(* CoDeSys 2.3.9.36 project: KVR_Mast.1.3.pro *)
(* Version: 13 *)
(* Author: JB *)
(* Libraries: ifm_CR0401\ifm_CR0401_V030100.lib 30.7.20 09:49:34, ifm_RAWCan\ifm_RAWCan_NT_V020004.lib 27.10.21 17:23:48, ifm_CANopen\ifm_CANopen_NT_V020004.lib 27.10.21 17:23:48, ifm_CANopen\3S_CanDrv.lib 27.10.21 17:23:48, ifm_CANopen\3S_CANopenManager.lib 27.10.21 17:23:48, Util.lib 6.11.07 14:39:24, standard.lib 4.10.05 11:14:46, SysLibCallback.lib 26.9.08 16:43:52 *)

(* PLC configuration (modules and I/O channels)
Configuration [LocalConfiguration] node 0, in %IB0 out %QB0 {IFM_PARAM_WORD_TIME = 0}
Input/Output [LocalInputOutput] node 1, in %IB0 out %QB0
IN00 AT %IB0 [ChInputBool] Input 00 Bit
IN01 AT %IB1 [ChInputBool] Input 01 Bit
IN02 AT %IB2 [ChInputBool] Input 02 Bit
IN03 AT %IB3 [ChInputBool] Input 03 Bit
IN04 AT %IB4 [ChInputBool] Input 04 Bit
IN05 AT %IB5 [ChInputBool] Input 05 Bit
IN06 AT %IB6 [ChInputBool] Input 06 Bit
IN07 AT %IB7 [ChInputBool] Input 07 Bit
IN08 AT %IB8 [ChInputBool] Input 08 Bit
IN09 AT %IB9 [ChInputBool] Input 09 Bit
IN10 AT %IB10 [ChInputBool] Input 10 Bit
IN11 AT %IB11 [ChInputBool] Input 11 Bit
OUT00 AT %QB0 [ChOutputBool] Output 00 Bit
OUT01 AT %QB1 [ChOutputBool] Output 01 Bit
OUT02 AT %QB2 [ChOutputBool] Output 02 Bit
OUT03 AT %QB3 [ChOutputBool] Output 03 Bit
OUT04 AT %QB4 [ChOutputBool] Output 04 Bit
OUT05 AT %QB5 [ChOutputBool] Output 05 Bit
OUT06 AT %QB6 [ChOutputBool] Output 06 Bit
OUT07 AT %QB7 [ChOutputBool] Output 07 Bit
System Inputs [LocalSystemInputs] node 2, in %IB12 out %QB8
  SUPPLY_VOLTAGE_VBBS AT %IW6 [ChInputWord] Supply voltage VBBS
  SUPPLY_VOLTAGE_VU AT %IW7 [ChInputWord] Supply voltage VU
  SUPPLY_VOLTAGE_VBB1 AT %IW8 [ChInputWord] Supply voltage VBB1
  SUPPLY_VOLTAGE_VBB2 AT %IW9 [ChInputWord] Supply voltage VBB2
  TEMPERATURE AT %IW10 [ChInputInt] Temperature
J1939 Interface [CAN_J1939] node 1, in %IB22 out %QB8
J1939 Interface [CAN_J1939] node 1, in %IB44 out %QB16
*)

(* Global variable list: Global_Constants *)
VAR_GLOBAL CONSTANT

	MAX_CTRLINDEX: BYTE := 0;

	SIMULATIONSMODUS: BOOL := FALSE;

	(* Flag positions for variable FlagsECU2PC *)
	ECU2PC_AllowRemote: INT := 3;
	ECU2PC_EmergencyStop: INT := 4;
	ECU2PC_RemoteAckn: INT := 6;
	ECU2PC_MainSwitch: INT := 7;

	(* Flag positions for variable FlagsPC2ECU *)
	PC2ECU_Remote: INT := 0;
	PC2ECU_BlackOut: INT := 1;
	PC2ECU_ResetMotorActiveTime: INT := 3;

	(* Flag positions for variables Mast[x].FlagsECU2PC *)
	ECU2PC_TopPosition: INT := 0;
	ECU2PC_BottomPosition: INT := 1;
	ECU2PC_MovingUp: INT := 2;
	ECU2PC_MovingDown: INT := 3;
	ECU2PC_LocalUp: INT := 4;
	ECU2PC_LocalDown: INT := 5;
	ECU2PC_LimitSwitch4m: INT := 7;
	ECU2PC_LimitSwitchBottom: INT := 8;
	ECU2PC_NotReadyToSwitchOn: INT := 9;
	ECU2PC_ParkPosition: INT := 10;
	ECU2PC_MontagePos: INT := 11;
	ECU2PC_LimitSwitchAufgerichtet: INT := 12;

	(* Flag positions for variables Mast[x].FlagsPC2ECU *)
	PC2ECU_MoveUp: INT := 0;
	PC2ECU_MoveDown: INT := 1;
	PC2ECU_SlowSpeed: INT := 2;

	(* Flag positions for variable Mast[x].ErrorECU2PC *)
	ECU2PC_ErrorFU: INT 					:= 0;
	ECU2PC_ErrorCanTimeout: INT 			:= 1;
	ECU2PC_ErrorMastSchrittkette: INT 		:= 4;

	QSCMD_NOP: BYTE				:= 0;
	QSCMD_CLEAR_ERROR: BYTE		:= 1;
	QSCMD_QUICK_STOP: BYTE		:= 113;
	QSCMD_HALT: BYTE			:= 114;
	QSCMD_VELOCITY_MODE: BYTE	:= 117; (* QSData0 = desired velocity *)
	QSCMD_ABS_POS_MODE: BYTE	:= 118; (* QSData0 = desired velocity, QSData1 = desired position *)

	(* Flag positions for FU statusword *)
	STAT_ENABLED: INT			:= 0;
	STAT_ERROR: INT				:= 1;
	STAT_WARNING: INT			:= 2;
	STAT_MOVING: INT			:= 3;
	STAT_REACHED: INT			:= 4;
	STAT_LIMIT: INT				:= 5;
	STAT_STOP_OR_HALT: INT		:= 11;

	FU1_POS_TO_MM: REAL 		:= 4.1114E-004;

	CAN_CHANNEL_HOST: BYTE 		:= 1;
	CAN_CHANNEL_LOCAL: BYTE 	:= 2;

	FU1_NODE_ID: BYTE			:= 127;

	MAX_CURRENT_HIST: WORD		:= 100;
	MAX_ERRORCODE_HIST: BYTE	:= 10;

END_VAR

(* Global variable list: Global_Variables *)
VAR_GLOBAL

	BlinkSlow: BOOL;

	MasterPresent: BOOL;

	inputs: TYPE_INPUTS;
	outputs: TYPE_OUTPUTS;

	canNodeFU1Present: BOOL;

	tasteAuf: BOOL;
	tasteAb: BOOL;
	tasteReset: BOOL;

	FlagsECU2PC: WORD			{parameter list=proc_vars_ecu [name=FlagsECU2PC 					index=16#3000 subindex=1 accessright="read only"] };
	FlagsPC2ECU: WORD			{parameter list=proc_vars_ecu [name=FlagsPC2ECU 					index=16#3000 subindex=2 accessright="write only"] };
	Windspeed: BYTE				{parameter list=proc_vars_ecu [name=Windspeed	 					index=16#3000 subindex=3 accessright="read only"] };
	CabinetTemperature: SINT	{parameter list=proc_vars_ecu [name=Temperature	 					index=16#3000 subindex=4 accessright="read only"] };
	ExtTemperature: SINT		{parameter list=proc_vars_ecu [name=ExtTemperature	 				index=16#3000 subindex=5 accessright="read only"] };
	IntVoltage: WORD			{parameter list=proc_vars_ecu [name=IntVoltage		 				index=16#3000 subindex=6 accessright="read only"] };

	Mast1Height: WORD			{parameter list=proc_vars_mast1 [name=Mast1Height 					index=16#3001 subindex=1 accessright="read only"] };
	Mast1FlagsECU2PC: WORD		{parameter list=proc_vars_mast1 [name=Mast1FlagsECU2PC 				index=16#3003 subindex=1 accessright="read only"] };
	Mast1FlagsPC2ECU: WORD		{parameter list=proc_vars_mast1 [name=Mast1FlagsPC2ECU 				index=16#3004 subindex=1 accessright="write only"] };
	Mast1Current: DINT			{parameter list=proc_vars_mast1 [name=Mast1Current 					index=16#3006 subindex=1 accessright="read only"] };
	Mast1ErrorECU2PC: WORD		{parameter list=proc_vars_mast1 [name=Mast1ErrorECU2PC				index=16#300D subindex=1 accessright="read only"] };
	Mast1FUErrorCode: WORD		{parameter list=proc_vars_mast1 [name=Mast1FUErrorCode				index=16#3010 subindex=1 accessright="read only"] };
	Mast1State: BYTE			{parameter list=proc_vars_mast1 [name=Mast1State					index=16#3012 subindex=1 accessright="read only"] };
	Mast1Speed: DINT			{parameter list=proc_vars_mast1 [name=Mast1Speed					index=16#3013 subindex=1 accessright="read only"] };

	(*
	Mast1TempPcbPower: WORD		{parameter list=proc_vars_mast1 [name=Mast1TempPcbPower				index=16#300A subindex=1 accessright="read only"] };
	Mast1TempPcbController: WORD{parameter list=proc_vars_mast1 [name=Mast1TempPcbController		index=16#300B subindex=1 accessright="read only"] };
	Mast1TempPcbAmplifier: WORD	{parameter list=proc_vars_mast1 [name=Mast1TempPcbAmplifier			index=16#300F subindex=1 accessright="read only"] };
	*)

	Mast1SetEncoderPW: DWORD	{parameter list=Parameters 		[name=Mast1SetEncoderPW				index=16#2014 subindex=1 accessright="read-write"] };

	Version: BYTE				{parameter list=version_info 	[name=Version						index=16#3020 subindex=1 accessright="read only"] };
	VersionDate: DWORD			{parameter list=version_info 	[name=VersionDate					index=16#3020 subindex=2 accessright="read only"] };

	Mast1MotorActiveTimeSeconds2: DWORD {parameter list=proc_vars_mast1 [name=Mast1MotorActiveTimeSeconds2 index=16#3014 subindex=1 accessright="read only"] };

	FU1_Current_Sim: DINT;

	FU1_Current_Hist: ARRAY[0..MAX_CURRENT_HIST] OF DINT;
	FU1_ErrorCode_Idx: BYTE;
	FU1_ErrorCode_Hist: ARRAY[0..MAX_ERRORCODE_HIST] OF INT;

END_VAR

VAR_GLOBAL RETAIN
	Mast1HeightRetain: WORD;
    NullfahrtErforderlich: BOOL;
END_VAR

(* Global variable list: Parameters *)
VAR_GLOBAL RETAIN
	SettingsPW: DWORD := 0	 					{parameter list=Parameters [name=SettingsPW					 	index=16#2000 subindex=12 accessright="read-write"] };
	(* 9000 *)
	Mast1TopPosition: WORD := 12000 				{parameter list=Parameters [name=Mast1TopPosition 				index=16#2006 subindex=1 accessright="read-write"] };
	Mast1BottomPosition: WORD := 2975			{parameter list=Parameters [name=Mast1BottomPosition			index=16#2007 subindex=1 accessright="read-write"] };
	Mast1VelocityNormal: INT := 2500			{parameter list=Parameters [name=Mast1VelocityNormal			index=16#200A subindex=1 accessright="read-write"] };
	Mast1VelocitySlow: INT := 500				{parameter list=Parameters [name=Mast1VelocitySlow				index=16#200B subindex=1 accessright="read-write"] };
	Mast1VelocityBottom: INT := 500				{parameter list=Parameters [name=Mast1VelocityBottom			index=16#200C subindex=1 accessright="read-write"] };
	Mast1BottomPositionOffset: WORD := 60		{parameter list=Parameters [name=Mast1BottomPositionOffset		index=16#200D subindex=1 accessright="read-write"] };
	Mast1CurrentLimitBottom: INT := 30			{parameter list=Parameters [name=Mast1CurrentLimitBottom		index=16#200E subindex=1 accessright="read-write"] };
	Mast1BottomLimitSwitchWindow: WORD := 50	{parameter list=Parameters [name=Mast1BottomLimitSwitchWindow	index=16#200F subindex=1 accessright="read-write"] };
	Mast1MontagePos: WORD := 3975 				{parameter list=Parameters [name=Mast1MontagePos 				index=16#2010 subindex=1 accessright="read-write"] };
	Mast1MotorActiveTimeSeconds: DWORD := 0		{parameter list=Parameters [name=Mast1MotorActiveTimeSeconds	index=16#2013 subindex=1 accessright="read-write"] };
	Mast1CurrentLimit: INT := 50				{parameter list=Parameters [name=Mast1CurrentLimit				index=16#2018 subindex=1 accessright="read-write"] };
	Mast1TopSettlingOffset: INT := 40			{parameter list=Parameters [name=Mast1TopSettlingOffset			index=16#2019 subindex=1 accessright="read-write"] };
END_VAR

(* Data type *)
TYPE TYPE_INPUTS :
	STRUCT
		TasteAusfahren: BOOL;
		TasteEinfahren: BOOL;
		TastePoweredByGenerator: BOOL;
		EndschalterNotantrieb: BOOL;
		EndschalterEingefahren: BOOL;
		EndschalterAufgerichtet: BOOL;
	END_STRUCT
END_TYPE

(* Data type *)
TYPE TYPE_OUTPUTS :
	STRUCT
		LEDAusgefahren: BOOL;
		LEDEingefahren: BOOL;
		LEDMontagePos: BOOL;
		RelaisMotorLeistung: BOOL;
		SchuetzGrundlast: BOOL;
	END_STRUCT
END_TYPE

(* POU PLC_PRG, FBD *)
PROGRAM PLC_PRG
VAR
	Init1: BOOL:=TRUE;
	CycleTime:DWORD;
	MaxCycleTime:DWORD;
	ResetMax:BOOL;
END_VAR
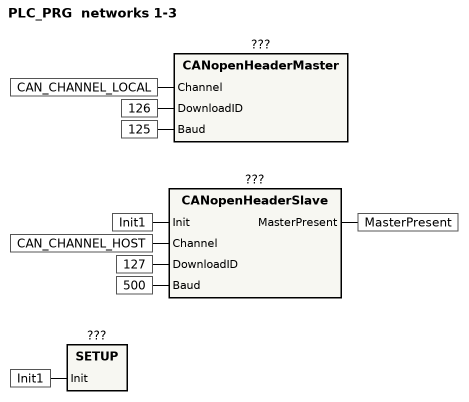
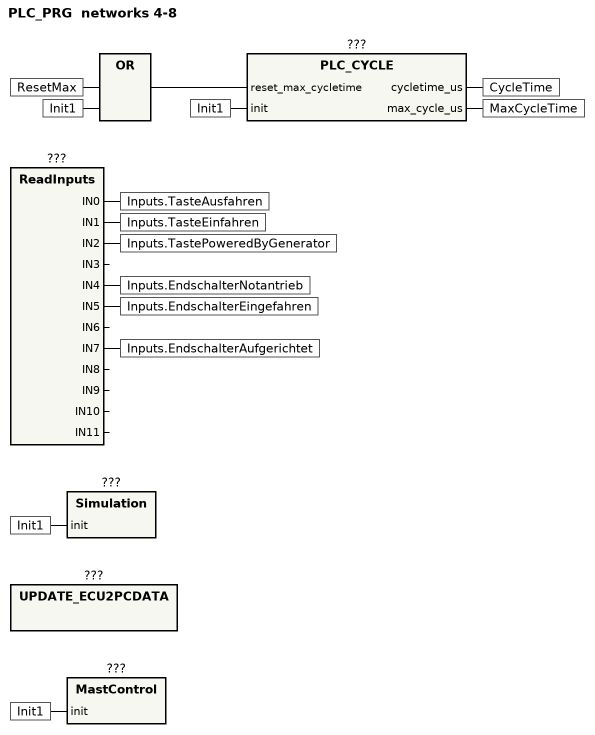
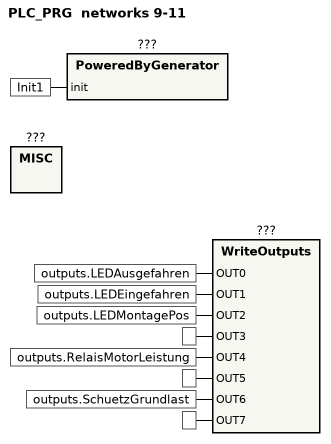
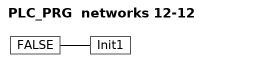
_FBD_ (* Function Block Diagram *)
NETWORK 1 (* CAN Master auf CAN2 initialisieren (Schnittstelle zu FU) *)
	???:CANopenHeaderMaster(Channel: CAN_CHANNEL_LOCAL, DownloadID: 126, Baud: 125)
NETWORK 2 (* CAN Slave auf CAN1 initialisieren (Schnittstelle zu PC) *)
	???:CANopenHeaderSlave(Init: Init1, Channel: CAN_CHANNEL_HOST, DownloadID: 127, Baud: 500) => MasterPresent
NETWORK 3
	???:SETUP(Init: Init1)
NETWORK 4
	???:PLC_CYCLE(reset_max_cycletime: OR(ResetMax, Init1), init: Init1, max_cycle_us => MaxCycleTime) => CycleTime
NETWORK 5
	???:ReadInputs(IN1 => Inputs.TasteEinfahren, IN2 => Inputs.TastePoweredByGenerator, IN4 => Inputs.EndschalterNotantrieb, IN5 => Inputs.EndschalterEingefahren, IN7 => Inputs.EndschalterAufgerichtet) => Inputs.TasteAusfahren
NETWORK 6
	???:Simulation(init: Init1)
NETWORK 7
	???:UPDATE_ECU2PCDATA()
NETWORK 8
	NOT ???:MastControl(init: Init1)
NETWORK 9
	???:PoweredByGenerator(init: Init1)
NETWORK 10
	???:MISC()
NETWORK 11
	???:WriteOutputs(OUT0: outputs.LEDAusgefahren, OUT1: outputs.LEDEingefahren, OUT2: outputs.LEDMontagePos, OUT3: , OUT4: outputs.RelaisMotorLeistung, OUT5: , OUT6: outputs.SchuetzGrundlast, OUT7: )
NETWORK 12 (* last line *)
	FALSE => Init1
_END_FBD_
(* the same logic as Structured Text *)
(* Network 1: see the listing above *)
(* Network 2: see the listing above *)
(* Network 3: see the listing above *)
(* Network 4: see the listing above *)
(* Network 5: see the listing above *)
(* Network 6: see the listing above *)
(* Network 7: see the listing above *)
(* Network 8: see the listing above *)
(* Network 9: see the listing above *)
(* Network 10: see the listing above *)
(* Network 11: see the listing above *)
(* Network 12 *)
Init1 := FALSE;
END_PROGRAM

(* POU CANopen/CANopenHeaderMaster, FBD *)
PROGRAM CANopenHeaderMaster
VAR_INPUT
	Channel: BYTE;
	DownloadID: BYTE;
	Baud: WORD;
END_VAR
VAR
	(*CAN settings*)
	SettingsCAN: CAN_SETTING_ST;

	(*Set CANopen state*)
	SetCanOpenState: CANOPEN_SETSTATE;
	SetState:BOOL:=TRUE;

	(*Handling CANopen status*)
	HandlingCANopen: CANopen_HANDLING_ST;
	Baudrate: DWORD;
	MasterState: BYTE;
	GuardError: BOOL;
	ErrorNodeList: ARRAY[0..MAXGUARDERR] OF BYTE;
	CanState: BYTE;
	Nodestate: BYTE;
	LastNodeState: BYTE;

	(*Emergency handling*)
	CanEmcy: CAN_EMCY;
	RestEmcyList: BOOL;
	EMCY_MSG_Count: DWORD; (* No of EMCY messages  Leaving errors are count too *)
	EmcyStruct: ARRAY[0..10] OF tT_EMCY;

	(*Handling CAN status*)
	StatusCan: CAN_Status_and_Errors;
	ResetCanFlags: BOOL;
	BusLoad: BYTE;
	BusOff: BOOL;
	RxOverflow: BOOL;
	RxWarning: BOOL;
	TxOverflow: BOOL;
	TxWarning: BOOL;

	GetstateSlave1: CANopen_GetStateSlave;

END_VAR
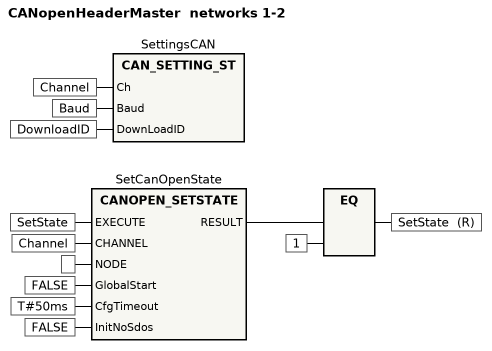
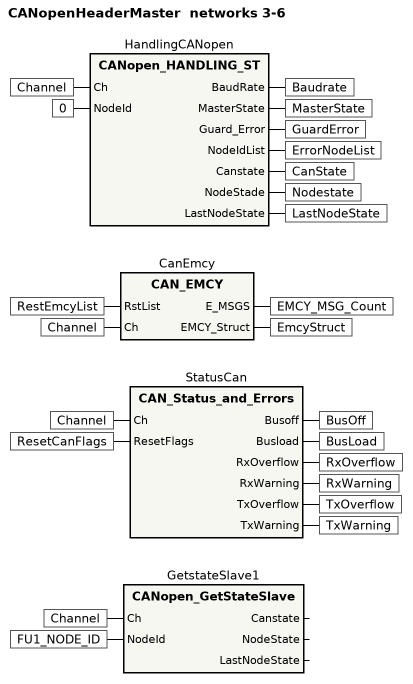
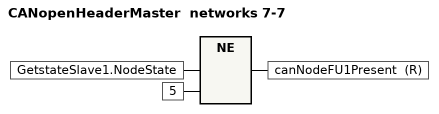
_FBD_ (* Function Block Diagram *)
NETWORK 1 (* Basic functions for the CAN / CANopen functionality *)
	SettingsCAN:CAN_SETTING_ST(Ch: Channel, Baud: Baud, DownLoadID: DownloadID)
NETWORK 2 (* Set CANopen status *)
	EQ(SetCanOpenState:CANOPEN_SETSTATE(EXECUTE: SetState, CHANNEL: Channel, NODE: , GlobalStart: FALSE, CfgTimeout: T#50ms, InitNoSdos: FALSE), 1) => R SetState
NETWORK 3 (* CANopen Master and heartbeat handling *)
	HandlingCANopen:CANopen_HANDLING_ST(Ch: Channel, NodeId: 0, MasterState => MasterState, Guard_Error => GuardError, NodeIdList => ErrorNodeList, Canstate => CanState, NodeStade => Nodestate, LastNodeState => LastNodeState) => Baudrate
NETWORK 4 (* CANopen Emergency Handling for 11 emergency messages *)
	CanEmcy:CAN_EMCY(RstList: RestEmcyList, Ch: Channel, EMCY_Struct => EmcyStruct) => EMCY_MSG_Count
NETWORK 5 (* Get the CAN Status and CAN Errors *)
	StatusCan:CAN_Status_and_Errors(Ch: Channel, ResetFlags: ResetCanFlags, Busload => BusLoad, RxOverflow => RxOverflow, RxWarning => RxWarning, TxOverflow => TxOverflow, TxWarning => TxWarning) => BusOff
NETWORK 6
	GetstateSlave1:CANopen_GetStateSlave(Ch: Channel, NodeId: FU1_NODE_ID)
NETWORK 7
	NE(GetstateSlave1.NodeState, 5) => R canNodeFU1Present
_END_FBD_
(* the same logic as Structured Text *)
(* Network 1 *)
SettingsCAN(Ch := Channel, Baud := Baud, DownLoadID := DownloadID);
(* Network 2: see the listing above *)
(* Network 3 *)
HandlingCANopen(Ch := Channel, NodeId := 0);
MasterState := HandlingCANopen.MasterState;
GuardError := HandlingCANopen.Guard_Error;
ErrorNodeList := HandlingCANopen.NodeIdList;
CanState := HandlingCANopen.Canstate;
Nodestate := HandlingCANopen.NodeStade;
LastNodeState := HandlingCANopen.LastNodeState;
Baudrate := HandlingCANopen.BaudRate;
(* Network 4 *)
CanEmcy(RstList := RestEmcyList, Ch := Channel);
EmcyStruct := CanEmcy.EMCY_Struct;
EMCY_MSG_Count := CanEmcy.E_MSGS;
(* Network 5 *)
StatusCan(Ch := Channel, ResetFlags := ResetCanFlags);
BusLoad := StatusCan.Busload;
RxOverflow := StatusCan.RxOverflow;
RxWarning := StatusCan.RxWarning;
TxOverflow := StatusCan.TxOverflow;
TxWarning := StatusCan.TxWarning;
BusOff := StatusCan.Busoff;
(* Network 6 *)
GetstateSlave1(Ch := Channel, NodeId := FU1_NODE_ID);
(* Network 7 *)
IF GetstateSlave1.NodeState <> 5 THEN canNodeFU1Present := FALSE; END_IF;
END_PROGRAM

(* POU CANopen/CAN_SETTING_ST, ST *)
FUNCTION_BLOCK CAN_SETTING_ST
(* Basic functions for the CAN / CANopen functionality *)
VAR

	CAN_SETDOWNLOADID_: CAN_SETDOWNLOADID;
	CAN_ENABLE_: CAN_ENABLE;
	CANOPEN_ENABLE_: CANOPEN_ENABLE;

	CANOPEN_SETSTATE_: CANOPEN_SETSTATE;
END_VAR
VAR_INPUT
	Ch: BYTE;
	Baud:WORD;
	DownLoadID:BYTE;
END_VAR
CAN_SETDOWNLOADID_(EXECUTE:=TRUE , CHANNEL:=Ch , DOWNLOAD_ID:=DownLoadID , RESULT=> );
CAN_ENABLE_(ENABLE:=TRUE , CHANNEL:=Ch , BAUDRATE:=Baud , RESULT=> );
CANOPEN_ENABLE_(ENABLE:=TRUE , CHANNEL:=Ch , Baudrate:=Baud , RESULT=> );
END_FUNCTION_BLOCK

(* POU CANopen/CANopen_HANDLING_ST, ST *)
FUNCTION_BLOCK CANopen_HANDLING_ST
(* CANopen Master and heartbeat handling *)
VAR
	CANOPEN_GETSTATE_: CANOPEN_GETSTATE;
	Execute_Getstate: BOOL := TRUE;
	CANOPEN_GETGUARDHBERRLIST_: CANOPEN_GETGUARDHBERRLIST;
	Execute_Guardlst: BOOL := TRUE;
	ResetErrorList: BOOL;
	PlcNodeId: BYTE;
	i: INT;
	GuardErrorCnt: WORD;
END_VAR
VAR_INPUT
	Ch: BYTE;
	NodeId: BYTE;
END_VAR
VAR_OUTPUT
	BaudRate: DWORD;
	MasterState: BYTE;
	Guard_Error: BOOL;
	NodeIdList: ARRAY[0..MAXGUARDERR] OF BYTE;
	Canstate: BYTE;
	NodeStade: BYTE;
	LastNodeState: BYTE;
END_VAR
(* ^^^^ Get the current state of the CANopen master ^^^^ *)
CANOPEN_GETSTATE_(
	EXECUTE:=Execute_Getstate ,
	CHANNEL:=Ch ,
	NODE:=NodeId ,
	MASTERSTATE=>MasterState ,
	PLCNODEID=>PlcNodeId ,
	PLCBAUDRATE=>BaudRate ,
	PLCVERSION=>,
	CANSTATE=>Canstate ,
	NODESTATE=>NodeStade ,
	LASTNODESTATE=>LastNodeState ,
	RESULT=> );

(* Values are valid now, function call can be stopped *)
IF CANOPEN_GETSTATE_.RESULT= 1 THEN
	Execute_Getstate:=FALSE;
END_IF

(* Function is passive, execute again *)
IF CANOPEN_GETSTATE_.RESULT= 0 THEN
	Execute_Getstate:=TRUE;
END_IF

(* ^^^^^ Get heartbeaterror or nodeguarding error ^^^^ *)
CANOPEN_GETGUARDHBERRLIST_(
	EXECUTE:=Execute_Guardlst ,
	CHANNEL:=Ch ,
	ResetList:=ResetErrorList ,
	N_NODES=>GuardErrorCnt,
	NODEID=>NodeIdList ,
	RESULT=> );

(* Values are valid now, function call can be stopped *)
IF CANOPEN_GETGUARDHBERRLIST_.RESULT= 1 THEN
	Execute_Guardlst:= FALSE;
END_IF

(* Function is passive, execute again *)
IF CANOPEN_GETGUARDHBERRLIST_.RESULT= 0 THEN
	Execute_Guardlst:= TRUE;
END_IF

(* An heartbeaterror has been appeared *)
IF CANOPEN_GETGUARDHBERRLIST_.N_NODES >0 THEN
	Guard_Error:=TRUE;
ELSE
	Guard_Error:=FALSE;
END_IF;

IF Ch = CAN_CHANNEL_LOCAL THEN

	canNodeFU1Present := TRUE;
	
	FOR i := 0 TO GuardErrorCnt DO
		IF FU1_NODE_ID = NodeIdList[i] THEN
			canNodeFU1Present := FALSE;
		END_IF
	END_FOR

END_IF
END_FUNCTION_BLOCK

(* POU CANopen/CAN_EMCY, FBD *)
FUNCTION_BLOCK CAN_EMCY
VAR_INPUT
	RstList: BOOL;
	Ch: BYTE;
END_VAR
VAR_OUTPUT
	E_MSGS: DWORD;
	EMCY_Struct: ARRAY[0..10] OF tT_EMCY;
END_VAR
VAR
	CANOPEN_GETEMCYMESSAGES_: CANOPEN_GETEMCYMESSAGES;
	Get_EMCY_MSG: BOOL := TRUE;
END_VAR
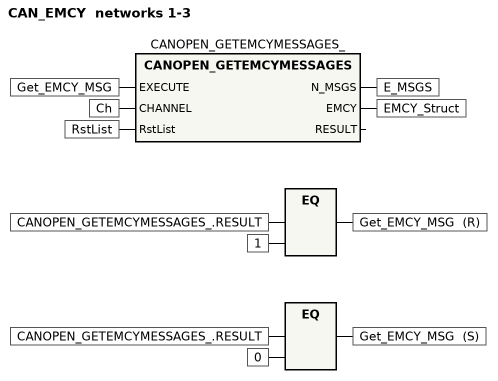
_FBD_ (* Function Block Diagram *)
NETWORK 1
	CANOPEN_GETEMCYMESSAGES_:CANOPEN_GETEMCYMESSAGES(EXECUTE: Get_EMCY_MSG, CHANNEL: Ch, RstList: RstList, EMCY => EMCY_Struct) => E_MSGS
NETWORK 2
	EQ(CANOPEN_GETEMCYMESSAGES_.RESULT, 1) => R Get_EMCY_MSG
NETWORK 3
	EQ(CANOPEN_GETEMCYMESSAGES_.RESULT, 0) => S Get_EMCY_MSG
_END_FBD_
(* the same logic as Structured Text *)
(* Network 1 *)
CANOPEN_GETEMCYMESSAGES_(EXECUTE := Get_EMCY_MSG, CHANNEL := Ch, RstList := RstList);
EMCY_Struct := CANOPEN_GETEMCYMESSAGES_.EMCY;
E_MSGS := CANOPEN_GETEMCYMESSAGES_.N_MSGS;
(* Network 2 *)
IF CANOPEN_GETEMCYMESSAGES_.RESULT = 1 THEN Get_EMCY_MSG := FALSE; END_IF;
(* Network 3 *)
IF CANOPEN_GETEMCYMESSAGES_.RESULT = 0 THEN Get_EMCY_MSG := TRUE; END_IF;
END_FUNCTION_BLOCK

(* POU CANopen/CAN_Status_and_Errors, FBD *)
FUNCTION_BLOCK CAN_Status_and_Errors
(* Get the CAN Status and CAN Errors *)
VAR

	CanStatus:CAN_STATUS;
	GETBUFFERFLAGS: CANOPEN_GETBUFFERFLAGS;

	ExecuteBufferFlags: BOOL:=TRUE;

END_VAR
VAR_INPUT
	Ch: BYTE;

	ResetFlags: BOOL;
END_VAR
VAR_OUTPUT
	Busoff: BOOL;
	Busload: BYTE;
	RxOverflow: BOOL;
	RxWarning: BOOL;
	TxOverflow: BOOL;
	TxWarning: BOOL;
END_VAR
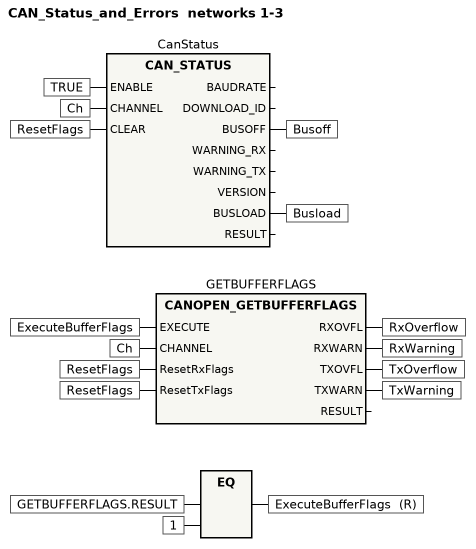
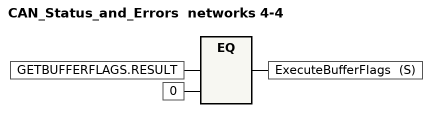
_FBD_ (* Function Block Diagram *)
NETWORK 1 (* Get the CAN Status *)
	CanStatus:CAN_STATUS(ENABLE: TRUE, CHANNEL: Ch, CLEAR: ResetFlags, BUSOFF => Busoff, BUSLOAD => Busload)
NETWORK 2 (* Get Buffer warnings / Reset Buffer Warning *)
	GETBUFFERFLAGS:CANOPEN_GETBUFFERFLAGS(EXECUTE: ExecuteBufferFlags, CHANNEL: Ch, ResetRxFlags: ResetFlags, ResetTxFlags: ResetFlags, RXWARN => RxWarning, TXOVFL => TxOverflow, TXWARN => TxWarning) => RxOverflow
NETWORK 3
	EQ(GETBUFFERFLAGS.RESULT, 1) => R ExecuteBufferFlags
NETWORK 4
	EQ(GETBUFFERFLAGS.RESULT, 0) => S ExecuteBufferFlags
_END_FBD_
(* the same logic as Structured Text *)
(* Network 1: Get the CAN Status *)
CanStatus(ENABLE := TRUE, CHANNEL := Ch, CLEAR := ResetFlags);
Busoff := CanStatus.BUSOFF;
Busload := CanStatus.BUSLOAD;
(* Network 2: Get Buffer warnings / Reset Buffer Warning *)
GETBUFFERFLAGS(EXECUTE := ExecuteBufferFlags, CHANNEL := Ch, ResetRxFlags := ResetFlags, ResetTxFlags := ResetFlags);
RxWarning := GETBUFFERFLAGS.RXWARN;
TxOverflow := GETBUFFERFLAGS.TXOVFL;
TxWarning := GETBUFFERFLAGS.TXWARN;
RxOverflow := GETBUFFERFLAGS.RXOVFL;
(* Network 3 *)
IF GETBUFFERFLAGS.RESULT = 1 THEN ExecuteBufferFlags := FALSE; END_IF;
(* Network 4 *)
IF GETBUFFERFLAGS.RESULT = 0 THEN ExecuteBufferFlags := TRUE; END_IF;
END_FUNCTION_BLOCK

(* POU CANopen/CANopen_GetStateSlave, ST *)
FUNCTION_BLOCK CANopen_GetStateSlave
VAR
	CANOPEN_GETSTATE_: CANOPEN_GETSTATE;
	Execute_Getstate: BOOL := TRUE;
END_VAR
VAR_INPUT
	Ch: BYTE;
	NodeId: BYTE;
END_VAR
VAR_OUTPUT
	Canstate: BYTE;
	NodeState: BYTE;
	LastNodeState: BYTE;
END_VAR
CANOPEN_GETSTATE_(
	EXECUTE:=Execute_Getstate ,
	CHANNEL:=Ch ,
	NODE:=NodeId ,
	MASTERSTATE=>,
	PLCNODEID=> ,
	PLCBAUDRATE=> ,
	PLCVERSION=>,
	CANSTATE=>Canstate ,
	NODESTATE=>NodeState ,
	LASTNODESTATE=>LastNodeState ,
	RESULT=> );

(* Values are valid now, function call can be stopped *)
IF CANOPEN_GETSTATE_.RESULT= 1 THEN
	Execute_Getstate:=FALSE;
END_IF

(* Function is passive, execute again *)
IF CANOPEN_GETSTATE_.RESULT= 0 THEN
	Execute_Getstate:=TRUE;
END_IF
END_FUNCTION_BLOCK

(* POU CANopen/CANopenHeaderSlave, FBD *)
PROGRAM CANopenHeaderSlave
VAR_INPUT
	Init: BOOL;
	Channel: BYTE;
	DownloadID: BYTE;
	Baud: WORD;
END_VAR
VAR_OUTPUT
	MasterPresent: BOOL;
END_VAR
VAR
	(*SettingsCAN*)
	SettingsCAN: CAN_SETTING_ST;

	(*Get status*)
	GetStateSlave: CANOPEN_GETNMTSTATESLAVE;
	SetGetStateSlave: BOOL;
	ResultState: BYTE;
	NodeState: BYTE;

	(*Get CANopen Node ID*)
	GetState: CANOPEN_GETSTATE;
	NodeId: BYTE;

	(*Get Guarding status*)
	GetGuard: CANOPEN_GETGUARDHBSTATSLV;
	GetGuardEx: BOOL;
	ResetGuard: BOOL;

END_VAR
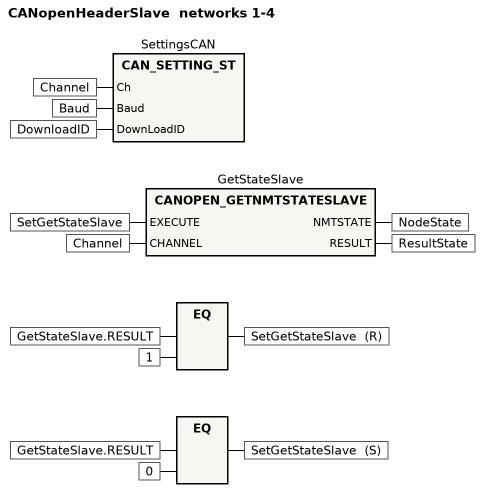
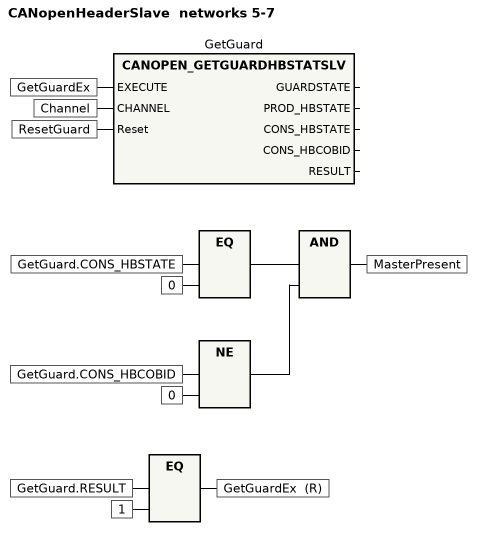
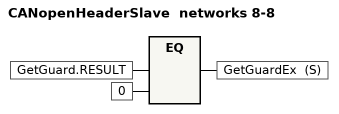
_FBD_ (* Function Block Diagram *)
NETWORK 1 (* Basic functions for the CAN / CANopen functionality *)
	SettingsCAN:CAN_SETTING_ST(Ch: Channel, Baud: Baud, DownLoadID: DownloadID)
NETWORK 2
	GetStateSlave:CANOPEN_GETNMTSTATESLAVE(EXECUTE: SetGetStateSlave, CHANNEL: Channel, RESULT => ResultState) => NodeState
NETWORK 3
	EQ(GetStateSlave.RESULT, 1) => R SetGetStateSlave
NETWORK 4
	EQ(GetStateSlave.RESULT, 0) => S SetGetStateSlave
NETWORK 5
	GetGuard:CANOPEN_GETGUARDHBSTATSLV(EXECUTE: GetGuardEx, CHANNEL: Channel, Reset: ResetGuard)
NETWORK 6
	AND(EQ(GetGuard.CONS_HBSTATE, 0), NE(GetGuard.CONS_HBCOBID, 0)) => MasterPresent
NETWORK 7
	EQ(GetGuard.RESULT, 1) => R GetGuardEx
NETWORK 8
	EQ(GetGuard.RESULT, 0) => S GetGuardEx
_END_FBD_
(* the same logic as Structured Text *)
(* Network 1: Basic functions for the CAN / CANopen functionality *)
SettingsCAN(Ch := Channel, Baud := Baud, DownLoadID := DownloadID);
(* Network 2 *)
GetStateSlave(EXECUTE := SetGetStateSlave, CHANNEL := Channel);
ResultState := GetStateSlave.RESULT;
NodeState := GetStateSlave.NMTSTATE;
(* Network 3 *)
IF GetStateSlave.RESULT = 1 THEN SetGetStateSlave := FALSE; END_IF;
(* Network 4 *)
IF GetStateSlave.RESULT = 0 THEN SetGetStateSlave := TRUE; END_IF;
(* Network 5 *)
GetGuard(EXECUTE := GetGuardEx, CHANNEL := Channel, Reset := ResetGuard);
(* Network 6 *)
MasterPresent := (GetGuard.CONS_HBSTATE = 0) AND (GetGuard.CONS_HBCOBID <> 0);
(* Network 7 *)
IF GetGuard.RESULT = 1 THEN GetGuardEx := FALSE; END_IF;
(* Network 8 *)
IF GetGuard.RESULT = 0 THEN GetGuardEx := TRUE; END_IF;
END_PROGRAM

(* POU Steuerung/SETUP, ST *)
PROGRAM SETUP
VAR_INPUT
	Init: BOOL;
END_VAR
VAR
	getAppInfo: GET_APP_INFO;
END_VAR
IF NOT Init THEN
	RETURN;
END_IF;

Mast1FlagsECU2PC.ECU2PC_ParkPosition := FALSE;

getAppInfo(ENABLE := TRUE);

VersionDate := STRING_TO_DWORD(LEFT(getAppInfo.BUILD_DATE, 8));
Version := STRING_TO_BYTE(LEFT(getAppInfo.VERSION, 3));
END_PROGRAM

(* POU PLC_CYCLE, ST *)
PROGRAM PLC_CYCLE
VAR_INPUT
	reset_max_cycletime: BOOL;
	init: BOOL;
END_VAR
VAR_OUTPUT
	cycletime_us: DWORD;
	max_cycle_us: DWORD;
END_VAR
VAR
	old_cycle: DWORD;
	TIMER_READ_US1: TIMER_READ_US;
	cycle: DWORD;
	nextTS: DWORD;
END_VAR
TIMER_READ_US1(TIME_US=>cycle );
cycletime_us:=cycle-old_cycle;
old_cycle:=cycle;

IF max_cycle_us<cycletime_us AND NOT init THEN
	max_cycle_us:=cycletime_us;
END_IF

IF reset_max_cycletime THEN
	max_cycle_us:=0;
END_IF

IF init THEN
	nextTS := cycle;
END_IF
(* Mehr als 1 Mio Ticks vergangen? *)
(* Zweikomplementarithmetik, d.h. funktioniert auch bei DWORD-Überlauf *)
IF cycle - nextTS > 1000000 THEN
	(* Das nächste Mal wieder nach 1 Mio Ticks (=1 Sekunde) *)
	nextTS := nextTS + 1000000;
	IF FU1_QSCmd <> QSCMD_HALT THEN
		Mast1MotorActiveTimeSeconds := Mast1MotorActiveTimeSeconds + 1;
	END_IF
END_IF
IF FlagsPC2ECU.PC2ECU_ResetMotorActiveTime THEN
	Mast1MotorActiveTimeSeconds := 0;
END_IF
END_PROGRAM

(* POU InputsOutputs/ReadInputs, FBD *)
PROGRAM ReadInputs
VAR
	_input: ARRAY[0..11] OF INPUT;
END_VAR
VAR_OUTPUT
	IN0: BOOL;
	IN1: BOOL;
	IN2: BOOL;
	IN3: BOOL;
	IN4: BOOL;
	IN5: BOOL;
	IN6: BOOL;
	IN7: BOOL;
	IN8: BOOL;
	IN9: BOOL;
	IN10: BOOL;
	IN11: BOOL;
END_VAR
VAR CONSTANT
	ModeInput_Off: BYTE := 0;
	ModeInput_0_10V: BYTE := 3;
	ModeInput_Ratio: BYTE := 6;
	ModeInput_0_20mA: BYTE := 7;
	ModeInput_0_32V: BYTE := 9;
	ModeInput_LowSide: BYTE := 10;
	ModeInput_LowSideNamur: BYTE := 11;
	ModeInput_HighSide: BYTE := 12;
	ModeInput_Resistor: BYTE := 18;
END_VAR
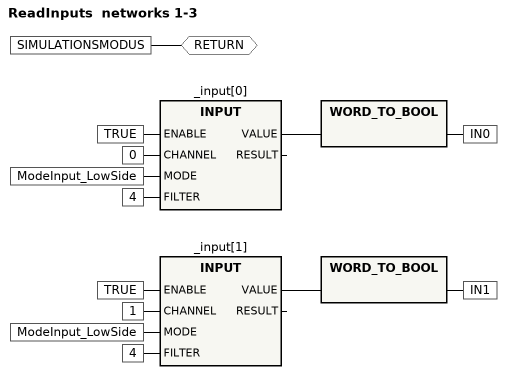
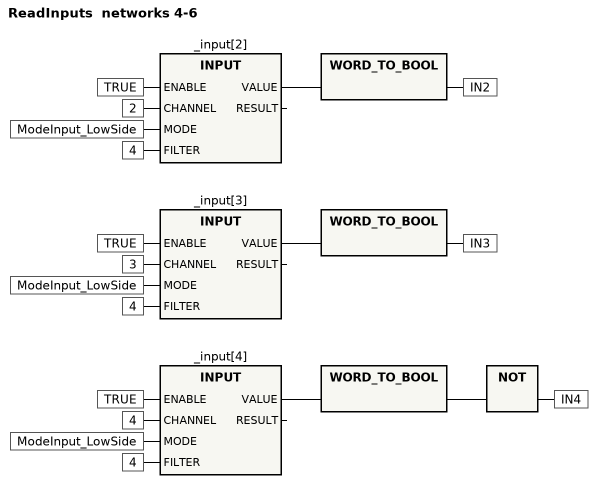
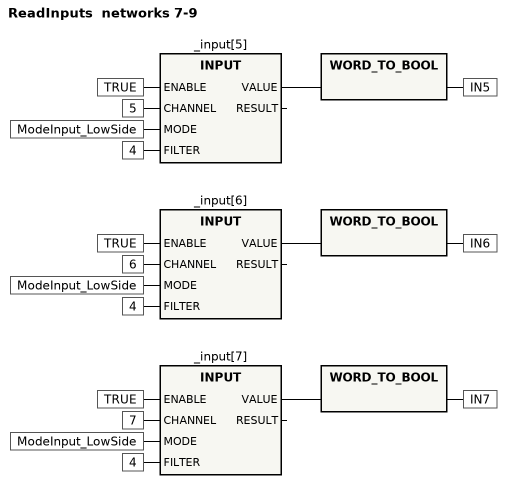
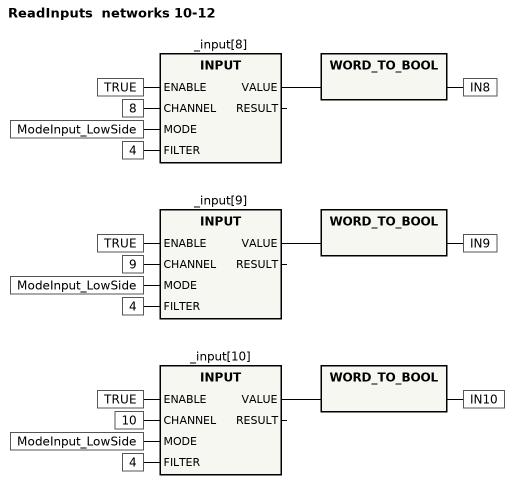
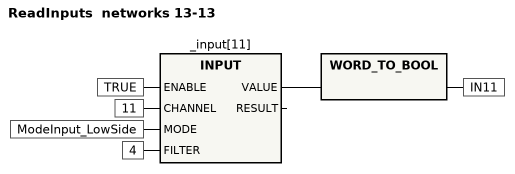
_FBD_ (* Function Block Diagram *)
NETWORK 1
	SIMULATIONSMODUS => <RETURN>
NETWORK 2
	WORD_TO_BOOL(_input[0]:INPUT(ENABLE: TRUE, CHANNEL: 0, MODE: ModeInput_LowSide, FILTER: 4)) => IN0
NETWORK 3
	WORD_TO_BOOL(_input[1]:INPUT(ENABLE: TRUE, CHANNEL: 1, MODE: ModeInput_LowSide, FILTER: 4)) => IN1
NETWORK 4
	WORD_TO_BOOL(_input[2]:INPUT(ENABLE: TRUE, CHANNEL: 2, MODE: ModeInput_LowSide, FILTER: 4)) => IN2
NETWORK 5
	WORD_TO_BOOL(_input[3]:INPUT(ENABLE: TRUE, CHANNEL: 3, MODE: ModeInput_LowSide, FILTER: 4)) => IN3
NETWORK 6
	NOT WORD_TO_BOOL(_input[4]:INPUT(ENABLE: TRUE, CHANNEL: 4, MODE: ModeInput_LowSide, FILTER: 4)) => IN4
NETWORK 7
	WORD_TO_BOOL(_input[5]:INPUT(ENABLE: TRUE, CHANNEL: 5, MODE: ModeInput_LowSide, FILTER: 4)) => IN5
NETWORK 8
	WORD_TO_BOOL(_input[6]:INPUT(ENABLE: TRUE, CHANNEL: 6, MODE: ModeInput_LowSide, FILTER: 4)) => IN6
NETWORK 9
	WORD_TO_BOOL(_input[7]:INPUT(ENABLE: TRUE, CHANNEL: 7, MODE: ModeInput_LowSide, FILTER: 4)) => IN7
NETWORK 10
	WORD_TO_BOOL(_input[8]:INPUT(ENABLE: TRUE, CHANNEL: 8, MODE: ModeInput_LowSide, FILTER: 4)) => IN8
NETWORK 11
	WORD_TO_BOOL(_input[9]:INPUT(ENABLE: TRUE, CHANNEL: 9, MODE: ModeInput_LowSide, FILTER: 4)) => IN9
NETWORK 12
	WORD_TO_BOOL(_input[10]:INPUT(ENABLE: TRUE, CHANNEL: 10, MODE: ModeInput_LowSide, FILTER: 4)) => IN10
NETWORK 13
	WORD_TO_BOOL(_input[11]:INPUT(ENABLE: TRUE, CHANNEL: 11, MODE: ModeInput_LowSide, FILTER: 4)) => IN11
_END_FBD_
(* the same logic as Structured Text *)
(* Network 1 *)
IF SIMULATIONSMODUS THEN RETURN; END_IF;
(* Network 2 *)
_input[0](ENABLE := TRUE, CHANNEL := 0, MODE := ModeInput_LowSide, FILTER := 4);
IN0 := WORD_TO_BOOL(_input[0].VALUE);
(* Network 3 *)
_input[1](ENABLE := TRUE, CHANNEL := 1, MODE := ModeInput_LowSide, FILTER := 4);
IN1 := WORD_TO_BOOL(_input[1].VALUE);
(* Network 4 *)
_input[2](ENABLE := TRUE, CHANNEL := 2, MODE := ModeInput_LowSide, FILTER := 4);
IN2 := WORD_TO_BOOL(_input[2].VALUE);
(* Network 5 *)
_input[3](ENABLE := TRUE, CHANNEL := 3, MODE := ModeInput_LowSide, FILTER := 4);
IN3 := WORD_TO_BOOL(_input[3].VALUE);
(* Network 6 *)
_input[4](ENABLE := TRUE, CHANNEL := 4, MODE := ModeInput_LowSide, FILTER := 4);
IN4 := NOT WORD_TO_BOOL(_input[4].VALUE);
(* Network 7 *)
_input[5](ENABLE := TRUE, CHANNEL := 5, MODE := ModeInput_LowSide, FILTER := 4);
IN5 := WORD_TO_BOOL(_input[5].VALUE);
(* Network 8 *)
_input[6](ENABLE := TRUE, CHANNEL := 6, MODE := ModeInput_LowSide, FILTER := 4);
IN6 := WORD_TO_BOOL(_input[6].VALUE);
(* Network 9 *)
_input[7](ENABLE := TRUE, CHANNEL := 7, MODE := ModeInput_LowSide, FILTER := 4);
IN7 := WORD_TO_BOOL(_input[7].VALUE);
(* Network 10 *)
_input[8](ENABLE := TRUE, CHANNEL := 8, MODE := ModeInput_LowSide, FILTER := 4);
IN8 := WORD_TO_BOOL(_input[8].VALUE);
(* Network 11 *)
_input[9](ENABLE := TRUE, CHANNEL := 9, MODE := ModeInput_LowSide, FILTER := 4);
IN9 := WORD_TO_BOOL(_input[9].VALUE);
(* Network 12 *)
_input[10](ENABLE := TRUE, CHANNEL := 10, MODE := ModeInput_LowSide, FILTER := 4);
IN10 := WORD_TO_BOOL(_input[10].VALUE);
(* Network 13 *)
_input[11](ENABLE := TRUE, CHANNEL := 11, MODE := ModeInput_LowSide, FILTER := 4);
IN11 := WORD_TO_BOOL(_input[11].VALUE);
END_PROGRAM

(* POU Steuerung/Simulation, ST *)
PROGRAM Simulation
VAR_INPUT
	init: BOOL;
END_VAR
VAR
	cnt: WORD;
	zielposition: WORD;
	aufgerichtet: BOOL := TRUE;
	notantrieb: BOOL := FALSE;
END_VAR
IF NOT SIMULATIONSMODUS THEN
	RETURN;
END_IF

IF init THEN
	Mast1Height := Mast1BottomPosition;
END_IF
(*
IF MastControl.status = MastControl.STATUS_WRITE_OFFSET THEN
	Mast1Height := Mast1BottomPosition + Mast1BottomLimitSwitchWindow;
END_IF
*)
FU1_Current_Sim := 0;

zielposition := REAL_TO_WORD(FU1_QSData1*FU1_POS_TO_MM);
inputs.EndschalterEingefahren := Mast1Height <= Mast1BottomPosition + Mast1BottomLimitSwitchWindow;
inputs.EndschalterAufgerichtet := aufgerichtet;
inputs.EndschalterNotantrieb := notantrieb;

IF FU1_QSCmd = QSCMD_ABS_POS_MODE THEN
	IF zielposition > Mast1Height THEN
		Mast1Height := Mast1Height + 1;
		FU1_Current_Sim := 10;
	END_IF
	IF zielposition < Mast1Height THEN
		Mast1Height := Mast1Height - 1;
		FU1_Current_Sim := 10;
	END_IF
ELSIF FU1_QSCmd = QSCMD_VELOCITY_MODE THEN
	IF cnt > 0 THEN
		cnt := cnt - 1;
	ELSE
		cnt := 10;
		Mast1Height := Mast1Height - 1;
	END_IF
	IF Mast1Height = Mast1BottomPosition THEN
		FU1_Current_Sim := 35;
	ELSE
		FU1_Current_Sim := 10;
	END_IF
END_IF
END_PROGRAM

(* POU Steuerung/UPDATE_ECU2PCDATA, ST *)
PROGRAM UPDATE_ECU2PCDATA
VAR
	Mast1Pos: BOOL;
	Mast1ontagePos: BOOL;
END_VAR
FlagsECU2PC.ECU2PC_AllowRemote := TRUE;
FlagsECU2PC.ECU2PC_EmergencyStop := Inputs.EndschalterNotantrieb;
FlagsECU2PC.ECU2PC_RemoteAckn := FALSE;
FlagsECU2PC.ECU2PC_MainSwitch := TRUE;

Mast1MotorActiveTimeSeconds2 := Mast1MotorActiveTimeSeconds;
Mast1State := MastControl.status;

(******************* ECU to PC flags *******************)
Mast1FlagsECU2PC.ECU2PC_TopPosition := (MastControl.status = MastControl.STATUS_AUSGEFAHREN);
Mast1FlagsECU2PC.ECU2PC_BottomPosition := (MastControl.status = MastControl.STATUS_EINGEFAHREN
	OR MastControl.status = MastControl.STATUS_NULLFAHRT_EINGEFAHREN);
Mast1FlagsECU2PC.ECU2PC_MovingUp :=
	FU1_QSCmd = QSCmd_ABS_POS_MODE AND Mast1Height < REAL_TO_WORD(FU1_QSData1*FU1_POS_TO_MM)
	OR
	FU1_QSCmd = QSCMD_VELOCITY_MODE AND FU1_QSData0*FU1_POS_TO_MM > 0;
Mast1FlagsECU2PC.ECU2PC_MovingDown :=
	FU1_QSCmd = QSCmd_ABS_POS_MODE AND Mast1Height > REAL_TO_WORD(FU1_QSData1*FU1_POS_TO_MM)
	OR
	FU1_QSCmd = QSCMD_VELOCITY_MODE AND FU1_QSData0*FU1_POS_TO_MM < 0;
Mast1FlagsECU2PC.ECU2PC_LocalUp := Inputs.TasteAusfahren;
Mast1FlagsECU2PC.ECU2PC_LocalDown := Inputs.TasteEinfahren;
Mast1FlagsECU2PC.ECU2PC_LimitSwitch4m := FALSE;
Mast1FlagsECU2PC.ECU2PC_LimitSwitchBottom := Inputs.EndschalterEingefahren;
Mast1FlagsECU2PC.ECU2PC_ParkPosition := Mast1FlagsECU2PC.ECU2PC_BottomPosition;
Mast1FlagsECU2PC.ECU2PC_MontagePos := (Mast1Height = Mast1MontagePos);
Mast1FlagsECU2PC.ECU2PC_LimitSwitchAufgerichtet := Inputs.EndschalterAufgerichtet;
END_PROGRAM

(* POU Steuerung/MastControl, ST *)
PROGRAM MastControl
VAR_INPUT
	init: BOOL;
END_VAR
VAR
	status: BYTE := STATUS_INIT;
	masthoeheReal: REAL;
	masthoeheSchleichfahrt: WORD;
	masthoeheEndschalter: WORD;
	masthoeheAbsetzen: WORD;
	mastPosGueltig: BOOL := FALSE;
	TSStart: DWORD;
	rtTasteReset: R_TRIG;
	rtSystemEin: R_TRIG;
	ftEndschalterEingefahren: F_TRIG;
	tonSystemEin: TON;
	tonKompressor: TON;
	tofInit: TOF;
	tonVelocityMode: TON;
	blnk: BLINK;
	SDOData: ARRAY[0..3] OF BYTE;
	SDOWriteOffset: CANOPEN_SDOWRITE;
	errorCode71x: BOOL;
	targetVelocity: INT;
	currentVelocity: INT;
	idxHist: WORD := 0;
	FU1_ErrorCode_Old: INT;
END_VAR
VAR CONSTANT
	_100ms: DWORD := 100000;
	STATUS_INIT: 					BYTE := 0;
	STATUS_WAIT_FOR_CAN_CLIENTS: 	BYTE := 10;
	STATUS_SETUP_OFFSET: 			BYTE := 11;
	STATUS_WRITE_OFFSET: 			BYTE := 12;
	STATUS_SUCCESS: 				BYTE := 15;
	STATUS_NULLFAHRT_AUSFAHREN: 	BYTE := 20;
	STATUS_NULLFAHRT_EINFAHREN: 	BYTE := 21;
	STATUS_NULLFAHRT_EINGEFAHREN:	BYTE := 22;
	STATUS_NULLPUNKT_SETZEN_INIT: 	BYTE := 30;
	STATUS_NULLPUNKT_SETZEN: 		BYTE := 31;
	STATUS_IDLE: 					BYTE := 50;
	STATUS_AUSFAHREN: 				BYTE := 60;
	STATUS_AUSFAHREN_ES_SUCHEN: 	BYTE := 61;
	STATUS_ABSETZEN_INIT:			BYTE := 63;
	STATUS_ABSETZEN: 				BYTE := 64;
	STATUS_AUSGEFAHREN: 			BYTE := 65;
	STATUS_AUSFAHREN_MONTAGE: 		BYTE := 66;
	STATUS_MONTAGEPOSITION: 		BYTE := 67;
	STATUS_EINFAHREN: 				BYTE := 70;
	STATUS_SCHLEICHFAHRT: 			BYTE := 72;
	STATUS_EINGEFAHREN: 			BYTE := 73;

	(* Ständige Überprüfungen *)
	STATUS_ERR_FU_TIMEOUT: 			BYTE := 100; (* FU nicht (mehr) online *)
	STATUS_ERR_CURRENT: 			BYTE := 101; (* Hoher Grenzwert Strom überschritten *)
	STATUS_ERR_FU: 					BYTE := 102; (* FU meldet Fehler *)
	STATUS_ERR_NOTANTRIEB:			BYTE := 103; (* Endschalter Notantrieb betätigt *)

	(* Fehlerzustände in Schrittkette *)
	(* Definitionen: *)
	(* Position U: Parameter Masthöhe untere Position *)
	(* Position E: Parameter Masthöhe untere Position + Parameter Fenster unterer Endschalter *)
	(* Position S: Parameter Masthöhe untere Position + Parameter Offset untere Position *)
	(* Position A: Parameter Masthöhe obere Position - Parameter Mast oben Absetzen Offset *)
	(* Position O: Parameter Masthöhe obere Position *)
	(* Es muss gelten: Position U < Position E < Position S < Position A < Position O *)
	STATUS_ERR_SET_FU_POS: 			BYTE := 110; (* Fehler beim Setzen der Nullposition im FU, FU-Position springt nicht auf eingestellten Wert *)
	STATUS_ERR_CURRENT_BOTTOM: 		BYTE := 111; (* Bei langsamer Fahrt niedriger Grenzwert Strom überschritten *)

	STATUS_ERR_ES_UNTEN_AUSFAHREN1:	BYTE := 120; (* Beim Ausfahren Endschalter suchen: Endschalter UNTEN unterhalb Position S nicht gefunden *)
	STATUS_ERR_ES_UNTEN_AUSFAHREN2:	BYTE := 121; (* Beim Ausfahren: Endschalter UNTEN oberhalb Position E betätigt *)
	STATUS_ERR_ES_FREIG_AUSFAHREN1:	BYTE := 123; (* Beim Ausfahren auf Position O: Endschalter AUFGERICHTET nicht mehr betätigt *)

	STATUS_ERR_ES_UNTEN_ABSETZEN:	BYTE := 130; (* Beim Einfahren in Position A: Endschalter UNTEN betätigt *)

	STATUS_ERR_ES_UNTEN_EINFAHREN1:	BYTE := 140; (* Beim Einfahren auf Position S: Endschalter UNTEN betätigt *)
	STATUS_ERR_ES_UNTEN_EINFAHREN2:	BYTE := 141; (* Bei Schleichfahrt auf Position U: Endschalter UNTEN nicht gefunden *)
	STATUS_ERR_ES_UNTEN_EINFAHREN3:	BYTE := 142; (* Bei Schleichfahrt auf Position U: Endschalter UNTEN unterhalb Position E nicht mehr betätigt *)

END_VAR
(******************* Diverse Timer und Flankenauswertungen *******************)
tonSystemEin(IN := TRUE, PT := T#1000ms);
tofInit(IN := init, PT := T#3s);
rtSystemEin(CLK := NOT tofInit.Q);
blnk(ENABLE := TRUE, TIMELOW := T#200ms, TIMEHIGH := T#200ms);
ftEndschalterEingefahren(CLK := inputs.EndschalterEingefahren);

(******************* Initialisierungen *******************)
outputs.RelaisMotorLeistung := FALSE;
FU1_QSCmd := QSCMD_HALT;
masthoeheSchleichfahrt := Mast1BottomPosition + Mast1BottomPositionOffset;
masthoeheEndschalter := Mast1BottomPosition + Mast1BottomLimitSwitchWindow;
masthoeheAbsetzen := Mast1TopPosition - Mast1TopSettlingOffset;

IF NOT SIMULATIONSMODUS THEN
	masthoeheReal := DINT_TO_REAL(FU1_Position) * FU1_POS_TO_MM;
	Mast1Height := REAL_TO_WORD(masthoeheReal);
	Mast1Current := FU1_Current/1000;
ELSE
	Mast1Current := FU1_Current_Sim;
END_IF
Mast1FUErrorCode := FU1_ErrorCode;
Mast1Speed := FU1_Velocity;

(******************* Taste Reset *******************)
rtTasteReset(CLK := tasteReset);
IF rtTasteReset.Q THEN
    Mast1ErrorECU2PC := 0;
    IF mastPosGueltig AND NOT NullfahrtErforderlich THEN
        Status := STATUS_IDLE;
    ELSE
        Status := STATUS_INIT;
    END_IF
END_IF


(******************* Flag Mast-Position korrekt falls Endschalter betätigt und Masthöhe plausibel *******************)
(******************* -> Fehlermeldung Masthöhe unterdrücken, keine Nullfahrt notwendig *******************)
IF rtSystemEin.Q THEN
	mastPosGueltig := inputs.EndschalterEingefahren AND ABS_DIFF(Mast1Height, Mast1BottomPosition) <= 2;
END_IF

(******************* Fehlermeldungen *******************)
IF NOT canNodeFU1Present AND NOT tofInit.Q AND NOT SIMULATIONSMODUS THEN
	Mast1ErrorECU2PC.ECU2PC_ErrorCanTimeout := TRUE;
	Status := STATUS_ERR_FU_TIMEOUT;
END_IF

(* Auswertung FU Fehlercode *)
(* -710 -> Position unbekannt *)
(* -711 -> Positionswert ungültig *)

IF FU1_ErrorCode <> FU1_ErrorCode_Old AND FU1_ErrorCode_Idx <= MAX_ERRORCODE_HIST THEN
	FU1_ErrorCode_Hist[FU1_ErrorCode_Idx] := FU1_ErrorCode;
	FU1_ErrorCode_Idx := FU1_ErrorCode_Idx + 1;
END_IF

errorCode71x := FU1_ErrorCode = -710 OR FU1_ErrorCode = -711;

IF canNodeFU1Present AND tonSystemEin.Q AND FU1_ErrorCode <> 0 THEN
	Mast1ErrorECU2PC.ECU2PC_ErrorFU := TRUE;
	Status := STATUS_ERR_FU;
	IF errorCode71x THEN
		mastPosGueltig := FALSE;
	END_IF
END_IF

(******************* Fehler *******************)
IF ABS(Mast1Current) > Mast1CurrentLimit AND Status <> STATUS_SCHLEICHFAHRT THEN
	Status := STATUS_ERR_CURRENT;
END_IF

(******************* Notantrieb/Handkurbel *******************)
IF inputs.EndschalterNotantrieb THEN
    Status := STATUS_ERR_NOTANTRIEB;
    mastPosGueltig := FALSE;
    NullfahrtErforderlich := TRUE;
END_IF


(******************* Schrittkette *******************)
CASE status OF
	STATUS_INIT:
		Status := STATUS_WAIT_FOR_CAN_CLIENTS;
		TSStart := PLC_CYCLE.cycle;

	STATUS_WAIT_FOR_CAN_CLIENTS:
		(* Warten bis FU online ist *)
		FU1_QSCmd := QSCMD_CLEAR_ERROR;
		IF canNodeFU1Present OR SIMULATIONSMODUS THEN
			Status := STATUS_SUCCESS;
			TSStart := PLC_CYCLE.cycle;
		ELSIF PLC_CYCLE.cycle - TSStart > 20*_100ms THEN
			Status := STATUS_ERR_FU_TIMEOUT;
		END_IF

	STATUS_SUCCESS:
        (* Erst mal 1s warten nachdem FU online ist *)
        IF PLC_CYCLE.cycle - TSStart > 10*_100ms THEN
            (* Falls Endschalter EIN und Position plausibel -> normal Starten mit Anzeige 'Eingefahren' *)
            IF inputs.EndschalterEingefahren AND ABS_DIFF(Mast1Height, Mast1BottomPosition) <= 2 THEN
                Status := STATUS_EINGEFAHREN;
                NullfahrtErforderlich := FALSE;
            ELSIF ABS_DIFF(Mast1Height, Mast1HeightRetain) <= 5 AND NOT NullfahrtErforderlich AND NOT inputs.EndschalterEingefahren THEN
                (* Falls geringe (5mm) Abweichung zwischen gemerkter und aktueller Position *)
				(* und nicht auf unterem Endschalter (bei unterem Endschalter immer Nullfahrt *)
				(* -> normal Starten *)
                Status := STATUS_IDLE;
            ELSE
                (* Sonst Nullfahrt nach oben bzw. unten *)
                IF inputs.EndschalterEingefahren THEN
                    Status := STATUS_NULLFAHRT_AUSFAHREN;
                ELSE
                    Status := STATUS_NULLFAHRT_EINFAHREN;
                END_IF
            END_IF
        END_IF


	STATUS_NULLFAHRT_AUSFAHREN:
		IF tasteAb THEN
 			Status := STATUS_NULLFAHRT_EINFAHREN;
		ELSIF tasteAuf THEN
			IF ftEndschalterEingefahren.Q THEN
				(* Fallende Flanke Endschalter unten, Nullpunkt setzen *)
				Status := STATUS_NULLPUNKT_SETZEN_INIT;
			ELSIF inputs.EndschalterEingefahren THEN
				(* Ausfahren im Geschwindigkeitsmodus *)
				(* Velocity mode: pos = auffahren, neg = einfahren oder umgekehrt je nach Vorzeichen Umrechnungsfaktor *)
				IF FU1_POS_TO_MM > 0 THEN
					targetVelocity := Mast1VelocityBottom;
				ELSE
					targetVelocity := -Mast1VelocityBottom;
				END_IF
				FU1_QSCmd := QSCMD_VELOCITY_MODE;
			END_IF
		END_IF

	STATUS_NULLFAHRT_EINFAHREN:
		IF tasteAuf THEN
 			Status := STATUS_NULLFAHRT_AUSFAHREN;
		ELSIF tonVelocityMode.Q AND NOT inputs.EndschalterEingefahren AND ABS(Mast1Current) > Mast1CurrentLimitBottom THEN
			(* Stromgrenzwert darf erst erreicht werden wenn unterer Endschalter betätigt, einschaltverzögert *)
			Status := STATUS_ERR_CURRENT_BOTTOM;
		ELSIF tasteAb THEN
			IF inputs.EndschalterEingefahren THEN
				(* Endschalter erreicht *)
				Status := STATUS_NULLFAHRT_EINGEFAHREN;
			ELSE
				(* Einfahren im Geschwindigkeitsmodus *)
				(* Velocity mode: pos = auffahren, neg = einfahren oder umgekehrt je nach Vorzeichen Umrechnungsfaktor *)
				IF FU1_POS_TO_MM > 0 THEN
					targetVelocity := -Mast1VelocityBottom;
				ELSE
					targetVelocity := Mast1VelocityBottom;
				END_IF
				FU1_QSCmd := QSCMD_VELOCITY_MODE;
			END_IF
		END_IF

	STATUS_NULLFAHRT_EINGEFAHREN:
		FU1_QSCmd := QSCMD_HALT;
		IF tasteAuf THEN
			Status := STATUS_NULLFAHRT_AUSFAHREN;
		END_IF

	STATUS_NULLPUNKT_SETZEN_INIT:
		(* Initialisierung Nullpunkt setzen, Mast stoppen *)
		status := STATUS_NULLPUNKT_SETZEN;
		TSStart := PLC_CYCLE.cycle;
		FU1_QSCmd := QSCMD_QUICK_STOP;

	STATUS_NULLPUNKT_SETZEN:
		(* Nach 500ms Nullpunkt in FU schreiben *)
		FU1_QSCmd := QSCMD_QUICK_STOP;
		IF PLC_CYCLE.cycle - TSStart > 5*_100ms THEN
			(* Masthöhe für Endschalter-Position in FU schreiben *)
			DWORD_TO_BYTES(
				dw := REAL_TO_DINT((masthoeheEndschalter)/FU1_POS_TO_MM),
				ll => SDOData[0],
				ml => SDOData[1],
				mh => SDOData[2],
				hh => SDOData[3]);
			TSStart := PLC_CYCLE.cycle;
			status := STATUS_WRITE_OFFSET;
		END_IF

    STATUS_WRITE_OFFSET:
        (* 500ms warten, dann prüfen ob Masthöhe Endschalter-Position entspricht *)
        IF PLC_CYCLE.cycle - TSStart > 5*_100ms THEN
            (* Fehlermeldung Mastposition zurücksetzen *)
            IF Mast1Height = masthoeheEndschalter OR SIMULATIONSMODUS THEN
                (* statusOffset := STATUS_SETUP_SAVE; 'save' nicht mehr an FU schicken *)
                status := STATUS_IDLE;
                mastPosGueltig := TRUE;
                NullfahrtErforderlich := FALSE;
            ELSE
                status := STATUS_ERR_SET_FU_POS;
                CASE SDOWriteOffset.RESULT OF
                    1: (* FB-Ausführung wurde ohne Fehler beendet, Daten sind gültig *)
                        Mast1SetEncoderPW := 102;
                    32: (* SDO-Übertragung abgebrochen von Client oder Server *)
                        Mast1SetEncoderPW := 103;
                    33: (* TIMEOUT ist abgelaufen *)
                        Mast1SetEncoderPW := 104;
                    242: (* Fehler: Einstellung ist nicht möglich *)
                        Mast1SetEncoderPW := 105;
                    ELSE
                        Mast1SetEncoderPW := 106;
                END_CASE
            END_IF
        END_IF


	STATUS_IDLE:
		(* Startpunkt für Mast auf/ab fahren *)
		IF tasteAuf THEN
            IF inputs.EndschalterEingefahren THEN
                Status := STATUS_AUSFAHREN_ES_SUCHEN;
			ELSIF inputs.EndschalterAufgerichtet THEN
	            Status := STATUS_AUSFAHREN;
	        ELSE
	            Status := STATUS_AUSFAHREN_MONTAGE;
			END_IF
        ELSIF tasteAb THEN
            IF NOT inputs.EndschalterAufgerichtet AND Mast1Height > masthoeheSchleichfahrt
                    OR inputs.EndschalterAufgerichtet AND Mast1Height > Mast1MontagePos THEN
                Status := STATUS_EINFAHREN;
            ELSIF NOT inputs.EndschalterAufgerichtet THEN
                Status := STATUS_SCHLEICHFAHRT;
            END_IF
        END_IF


	STATUS_AUSFAHREN, STATUS_AUSFAHREN_ES_SUCHEN:
		IF NOT tasteAuf THEN
			(* Taste nicht mehr gedrückt? *)
			Status := STATUS_IDLE;
		ELSIF status = STATUS_AUSFAHREN_ES_SUCHEN AND Mast1Height >= masthoeheSchleichfahrt THEN
			(* Endschalter unten AUS oberhalb Position Schleichfahrt *)
			Status := STATUS_ERR_ES_UNTEN_AUSFAHREN1;
		ELSIF status = STATUS_AUSFAHREN_ES_SUCHEN AND NOT inputs.EndschalterEingefahren THEN
			(* Endschalter unten erreicht -> Nullpunkt setzen *)
			Status := STATUS_NULLPUNKT_SETZEN_INIT;
		ELSIF status = STATUS_AUSFAHREN AND inputs.EndschalterEingefahren THEN
			(* Endschalter unten EIN oberhalb Position Endschalter *)
			Status := STATUS_ERR_ES_UNTEN_AUSFAHREN2;
		ELSIF status = STATUS_AUSFAHREN AND NOT inputs.EndschalterAufgerichtet THEN
			(* Endschalter aufgerichtet AUS bei Fahrt auf obere Position *)
			Status := STATUS_ERR_ES_FREIG_AUSFAHREN1;
		ELSIF Mast1Height >= Mast1TopPosition THEN
			(* Obere Position erreicht -> Absetzen *)
			Status := STATUS_ABSETZEN_INIT;
		ELSE
			(* Bei Suche ES langsam fahren, sonst normale Geschwindigkeit *)
			IF status = STATUS_AUSFAHREN THEN
				IF Mast1FlagsPC2ECU.PC2ECU_SlowSpeed THEN
					FU1_QSData0 := Mast1VelocitySlow;
				ELSE
					FU1_QSData0 := Mast1VelocityNormal;
				END_IF
			ELSE
				FU1_QSData0 := Mast1VelocityBottom;
			END_IF
			(* Positionieren auf obere Position *)
			FU1_QSData1 := REAL_TO_DINT(WORD_TO_REAL(Mast1TopPosition)/FU1_POS_TO_MM);
			FU1_QSCmd := QSCMD_ABS_POS_MODE;
		END_IF

	STATUS_ABSETZEN_INIT:
		Status := STATUS_ABSETZEN;
		TSStart := PLC_CYCLE.cycle;

	STATUS_ABSETZEN:
		(* Automatische Fahrt, Taste nicht abfragen *)
		IF inputs.EndschalterEingefahren THEN
			(* Endschalter unten EIN bei Fahrt auf Absetzposition *)
			Status := STATUS_ERR_ES_UNTEN_ABSETZEN;
		ELSIF Mast1Height <= masthoeheAbsetzen THEN
			(* Absetzposition erreicht *)
			Status := STATUS_AUSGEFAHREN;
		ELSE
			(* Positionieren auf Absetzposition mit Geschwindigkeit Schleichfahrt *)
			FU1_QSData0 := Mast1VelocityBottom;
			FU1_QSData1 := REAL_TO_DINT(WORD_TO_REAL(masthoeheAbsetzen)/FU1_POS_TO_MM);
			FU1_QSCmd := QSCMD_ABS_POS_MODE;
		END_IF

	STATUS_AUSGEFAHREN:
		IF tasteAb THEN
			Status := STATUS_IDLE;
		END_IF

	STATUS_AUSFAHREN_MONTAGE:
		IF NOT tasteAuf THEN
			(* Taste nicht mehr gedrückt? *)
			Status := STATUS_IDLE;
		ELSIF inputs.EndschalterEingefahren THEN
			(* Endschalter EIN oberhalb Höhe Endschalter *)
			Status := STATUS_ERR_ES_UNTEN_AUSFAHREN2;
		ELSIF Mast1Height >= Mast1MontagePos THEN
			(* Montageposition erreicht *)
			Status := STATUS_MONTAGEPOSITION;
		ELSE
			(* Positionieren auf Montageposition mit normaler Geschwindigkeit *)
			IF Mast1FlagsPC2ECU.PC2ECU_SlowSpeed THEN
				FU1_QSData0 := Mast1VelocitySlow;
			ELSE
				FU1_QSData0 := Mast1VelocityNormal;
			END_IF
			FU1_QSData1 := REAL_TO_DINT(WORD_TO_REAL(Mast1MontagePos)/FU1_POS_TO_MM);
			FU1_QSCmd := QSCMD_ABS_POS_MODE;
		END_IF

	STATUS_MONTAGEPOSITION:
		IF tasteAb THEN
			Status := STATUS_IDLE;
		ELSIF tasteAuf AND inputs.EndschalterAufgerichtet THEN
			Status := STATUS_IDLE;
		END_IF


	STATUS_EINFAHREN:
        IF NOT tasteAb THEN
            (* Taste nicht mehr gedrückt? *)
            Status := STATUS_IDLE;
        ELSIF inputs.EndschalterEingefahren THEN
            (* Endschalter unten EIN oberhalb Position Schleichfahrt *)
            Status := STATUS_ERR_ES_UNTEN_EINFAHREN1;
        ELSIF inputs.EndschalterAufgerichtet THEN
            IF Mast1Height <= Mast1MontagePos THEN
                (* Position Montage erreicht *)
                Status := STATUS_IDLE;
            ELSE
                (* Positionieren auf Position Montage mit normaler Geschwindigkeit *)
                IF Mast1FlagsPC2ECU.PC2ECU_SlowSpeed THEN
                    FU1_QSData0 := Mast1VelocitySlow;
                ELSE
                    FU1_QSData0 := Mast1VelocityNormal;
                END_IF
                FU1_QSData1 := REAL_TO_DINT(WORD_TO_REAL(Mast1MontagePos)/FU1_POS_TO_MM);
                FU1_QSCmd := QSCMD_ABS_POS_MODE;
            END_IF
        ELSE
            IF Mast1Height <= masthoeheSchleichfahrt THEN
                (* Position Schleichfahrt erreicht *)
                Status := STATUS_IDLE;
            ELSE
                (* Positionieren auf Position Schleichfahrt mit normaler Geschwindigkeit *)
                IF Mast1FlagsPC2ECU.PC2ECU_SlowSpeed THEN
                    FU1_QSData0 := Mast1VelocitySlow;
                ELSE
                    FU1_QSData0 := Mast1VelocityNormal;
                END_IF
                FU1_QSData1 := REAL_TO_DINT(WORD_TO_REAL(masthoeheSchleichfahrt)/FU1_POS_TO_MM);
                FU1_QSCmd := QSCMD_ABS_POS_MODE;
            END_IF
        END_IF


	STATUS_SCHLEICHFAHRT:
		IF NOT tasteAb THEN
			(* Taste nicht mehr gedrückt? *)
			Status := STATUS_IDLE;
		ELSIF ABS(Mast1Current) > Mast1CurrentLimitBottom THEN
			Status := STATUS_ERR_CURRENT_BOTTOM;
	    ELSIF Mast1Height <= Mast1BottomPosition THEN
			(* Untere Position erreicht *)
			IF inputs.EndschalterEingefahren THEN
				Status := STATUS_EINGEFAHREN;
			ELSE
				(* Endschalter unten nicht erreicht *)
				Status := STATUS_ERR_ES_UNTEN_EINFAHREN2;
			END_IF
		ELSE
			(* Positionieren auf untere Position mit langsamer Geschwindigkeit *)
			FU1_QSData0 := Mast1VelocityBottom;
			FU1_QSData1 := REAL_TO_DINT(WORD_TO_REAL(Mast1BottomPosition)/FU1_POS_TO_MM);
			FU1_QSCmd := QSCMD_ABS_POS_MODE;
		END_IF

	STATUS_EINGEFAHREN:
		IF tasteAuf THEN
			Status := STATUS_IDLE;
		END_IF

END_CASE

(***** Aktuelle Masthöhe speichern falls Mast nicht in Initialisierungsphase/Nullfahrt *****)
IF Status >= STATUS_IDLE AND Mast1Height >= Mast1BottomPosition - 40 AND Mast1Height <= Mast1TopPosition + 10 THEN
	Mast1HeightRetain := Mast1Height;
END_IF

(******************* Schrittkette in Fehlerzustand *******************)
Mast1ErrorECU2PC.ECU2PC_ErrorMastSchrittkette := (Status >= 100);

(******************* FU-Fehler zurücksetzen *******************)
IF tasteReset (* OR errorCode71x *) (* OR NOT tonSystemEin.Q AND blnk.OUT*) THEN
	FU1_QSCmd := QSCMD_CLEAR_ERROR;  
END_IF

(******************* K1 Versorgung Motor *******************)
IF NOT inputs.EndschalterNotantrieb THEN
	outputs.RelaisMotorLeistung := TRUE;
END_IF

(******************* Rampe Geschwindigkeitsmodus *******************)
(* Nur beim Beschleunigen, beim Abbremsen soll sofort abgeschaltet werden *)
IF FU1_QSCmd = QSCMD_VELOCITY_MODE THEN
	IF targetVelocity > 0 THEN
		(* Positive Sollgeschwindigkeit: *)
		(* In jedem Zyklus 10 hochzählen bis Sollgeschwindigkeit erreicht *)
		(* D.h. bei 10ms Zykluszeit sind 500 U/min in 500ms erreicht*)
		currentVelocity := MIN(currentVelocity + 1, targetVelocity);
	ELSE
		(* Negative Sollgeschwindigkeit: *)
		(* In jedem Zyklus 10 runterzählen bis Sollgeschwindigkeit erreicht *)
		(* D.h. bei 10ms Zykluszeit sind 500 U/min in 500ms erreicht*)
		currentVelocity := MAX(currentVelocity - 1, targetVelocity);
	END_IF
	(* Geschwindigkeit setzen *)
	FU1_QSData0 := currentVelocity;
ELSE
	(* Auf 0 setzen falls kein Geschwindigkeitsmodus *)
	currentVelocity := 0;
END_IF

(******************* Einschaltverzögerung Geschwindigkeitsmodus *******************)
tonVelocityMode(IN := (FU1_QSCmd = QSCMD_VELOCITY_MODE), PT := T#1ms);

(******************* Nach Start im Geschwindigkeitsmodus die ersten 100 Stromwerte in Array schreiben *******************)
IF FU1_QSCmd = QSCMD_VELOCITY_MODE THEN
	IF idxHist <= MAX_CURRENT_HIST THEN
		FU1_Current_Hist[idxHist] := Mast1Current;
		idxHist := idxHist + 1;
	END_IF
ELSE
	idxHist := 0;
END_IF

(******************* SDO-Befehle *******************)
SDOWriteOffset(
	EXECUTE := status = STATUS_WRITE_OFFSET,
	CHANNEL := CAN_CHANNEL_LOCAL,
	NODE := FU1_NODE_ID,
	IDX := 16#4762,
	SUBIDX := 1,
	LEN := 4,
	DATA := SDOData,
	Timeout := T#200ms,
	RESULT => );
END_PROGRAM

(* POU Misc/ABS_DIFF, ST *)
FUNCTION ABS_DIFF : INT
VAR_INPUT
	A: WORD;
	B: WORD;
END_VAR
ABS_DIFF := ABS(WORD_TO_INT(A) - WORD_TO_INT(B));
END_FUNCTION

(* POU Misc/DWORD_TO_BYTES, ST *)
PROGRAM DWORD_TO_BYTES
VAR_INPUT
	dw: DWORD;
END_VAR
VAR_OUTPUT
	ll: BYTE;
	ml: BYTE;
	mh: BYTE;
	hh: BYTE;
END_VAR
ll := DWORD_TO_BYTE(dw);
ml := DWORD_TO_BYTE(SHR(dw, 8));
mh := DWORD_TO_BYTE(SHR(dw, 16));
hh := DWORD_TO_BYTE(SHR(dw, 24));
END_PROGRAM

(* POU Steuerung/PoweredByGenerator, ST *)
PROGRAM PoweredByGenerator
VAR_INPUT
	init: BOOL;
END_VAR
VAR
	rtTaste: R_TRIG;
	tofTaste: TOF;
END_VAR
IF init THEN
	(* Nach dem Einschalten erst mal aktivieren *)
	outputs.SchuetzGrundlast := TRUE;
END_IF

(* Taste entprellen *)
tofTaste(IN := inputs.TastePoweredByGenerator, PT := T#200ms);
rtTaste(CLK := tofTaste.Q);
IF rtTaste.Q THEN
	(* toggle *)
	outputs.SchuetzGrundlast := NOT outputs.SchuetzGrundlast;
END_IF
END_PROGRAM

(* POU Steuerung/MISC, ST *)
PROGRAM MISC
VAR
	TONInst: TON;
	OtherError: BOOL;
	TOFReset: TOF;
END_VAR
TONInst(IN := NOT TONInst.Q, PT:= T#500ms);
IF TONInst.Q THEN
	BlinkSlow := NOT BlinkSlow;
END_IF

IF NOT MasterPresent THEN
	FlagsPC2ECU := 0;
	Mast1FlagsPC2ECU := 0;
END_IF

IF Mast1ErrorECU2PC <> 0 OR MastControl.status >= 100 THEN
	Outputs.LEDAusgefahren := BlinkSlow;
	Outputs.LEDEingefahren := NOT BlinkSlow;
ELSE
	Outputs.LEDAusgefahren := Mast1FlagsECU2PC.ECU2PC_TopPosition;
	Outputs.LEDEingefahren := Mast1FlagsECU2PC.ECU2PC_ParkPosition;
END_IF

Outputs.LEDMontagePos := Mast1FlagsECU2PC.ECU2PC_MontagePos;

IntVoltage := SUPPLY_VOLTAGE_VBBS;

tasteReset := (tasteAuf AND tasteAb);
TOFReset(IN := tasteReset, PT := T#500ms);
tasteAuf := NOT TOFReset.Q AND (inputs.TasteAusfahren OR Mast1FlagsPC2ECU.PC2ECU_MoveUp);
tasteAb := NOT TOFReset.Q AND (inputs.TasteEinfahren OR Mast1FlagsPC2ECU.PC2ECU_MoveDown);
END_PROGRAM

(* POU InputsOutputs/WriteOutputs, FBD *)
PROGRAM WriteOutputs
VAR_INPUT
	OUT0: BOOL;
	OUT1: BOOL;
	OUT2: BOOL;
	OUT3: BOOL;
	OUT4: BOOL;
	OUT5: BOOL;
	OUT6: BOOL;
	OUT7: BOOL;
END_VAR
VAR
	_output: ARRAY[0..7] OF OUTPUT;
END_VAR
VAR CONSTANT
	ModeOutput_Off: BYTE := 0;
	ModeOutput_HighSide: BYTE := 2;
	ModeOutput_HighSide_Diag: BYTE := 15;
	ModeOutput_HighSide_Diag_Protection: BYTE := 16;
END_VAR
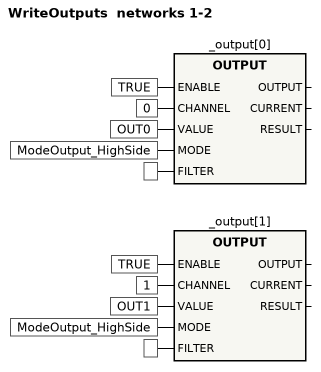
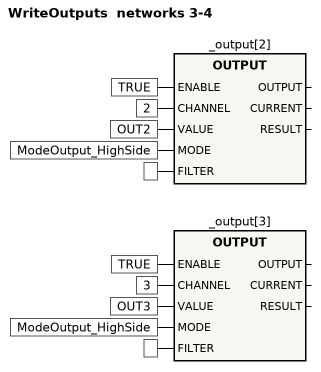
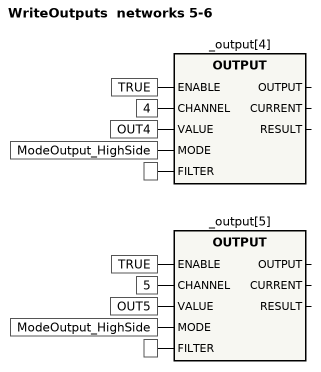
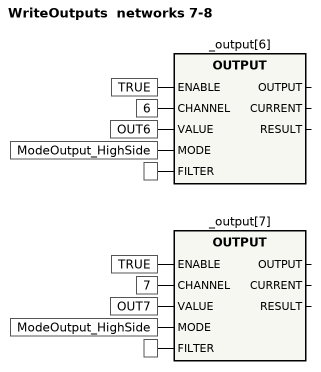
_FBD_ (* Function Block Diagram *)
NETWORK 1
	_output[0]:OUTPUT(ENABLE: TRUE, CHANNEL: 0, VALUE: OUT0, MODE: ModeOutput_HighSide, FILTER: )
NETWORK 2
	_output[1]:OUTPUT(ENABLE: TRUE, CHANNEL: 1, VALUE: OUT1, MODE: ModeOutput_HighSide, FILTER: )
NETWORK 3
	_output[2]:OUTPUT(ENABLE: TRUE, CHANNEL: 2, VALUE: OUT2, MODE: ModeOutput_HighSide, FILTER: )
NETWORK 4
	_output[3]:OUTPUT(ENABLE: TRUE, CHANNEL: 3, VALUE: OUT3, MODE: ModeOutput_HighSide, FILTER: )
NETWORK 5
	_output[4]:OUTPUT(ENABLE: TRUE, CHANNEL: 4, VALUE: OUT4, MODE: ModeOutput_HighSide, FILTER: )
NETWORK 6
	_output[5]:OUTPUT(ENABLE: TRUE, CHANNEL: 5, VALUE: OUT5, MODE: ModeOutput_HighSide, FILTER: )
NETWORK 7
	_output[6]:OUTPUT(ENABLE: TRUE, CHANNEL: 6, VALUE: OUT6, MODE: ModeOutput_HighSide, FILTER: )
NETWORK 8
	_output[7]:OUTPUT(ENABLE: TRUE, CHANNEL: 7, VALUE: OUT7, MODE: ModeOutput_HighSide, FILTER: )
_END_FBD_
END_PROGRAM
